FUNCTION_BLOCK FB_DefGridParamMediator IMPLEMENTS I_ParamMediator
VAR
  _pCamWorker : POINTER TO FB_WorkerDefGrid_Camera;
  _pDefWorker : POINTER TO FB_WorkerDefGrid_Deformation;
  bInitOk     : BOOL;
END_VAR

METHOD init
VAR_INPUT
  pCamWorker : POINTER TO FB_WorkerDefGrid_Camera;
  pDefWorker : POINTER TO FB_WorkerDefGrid_Deformation;
END_VAR
IF pCamWorker <> 0 AND pCamWorker <> 0 THEN
  _pCamWorker := pCamWorker;
  _pDefWorker := pDefWorker;
  bInitOk := TRUE;
END_IF
END_METHOD

PROPERTY sCameraGridSettings : ST_CameraGridSettings
GET
IF bInitOk THEN
  sCameraGridSettings := _pCamWorker^.sCameraGridSettings;
END_IF
END_GET
END_PROPERTY

PROPERTY sDeformationGridSetttings : ST_DefGridSettings
GET
IF bInitOk THEN
  sDeformationGridSetttings := _pDefWorker^.sDeformationGridSettings;
END_IF
END_GET
END_PROPERTY

END_FUNCTION_BLOCK

(* stored: Version 1.1.0.1, ProductVersion 3.1.4024.11
   POU FB_DefGridParamMediator: Id {9642270e-d441-4770-907b-3f0d0f5dc2e9}, SpecialFunc None
   Folder I_ParamMediator: Id {39f9222d-d28f-4df1-8ed1-e2b3d113f34f}
   Method init: Id {9cdfcac0-144a-4d88-8e7f-21c6ce0c82c3}
   Property sCameraGridSettings: Id {686354aa-821c-4c68-8c9d-dafadf8ef6fd}
   Get Get: Id {7a8afb02-f662-4c02-aebf-6b3bd22fae1a}
   Property sDeformationGridSetttings: Id {9cf3f096-207d-452b-ace7-3769f0678220}
   Get Get: Id {f92cba8c-0a7c-4567-a017-f6ac55645e3a} *)
